// TIA Portal V15.1 export
// export: Created 2026-01-15T16:29:37.3417303Z, ExportSetting WithDefaults, WithReadOnly, DisplayName Totally Integrated Automation Portal, DisplayVersion V15.1 Update 8, DisplayName TIA Portal Openness, DisplayVersion V15.1 Update 8, DisplayName STEP 7 Professional, DisplayVersion V15.1 Update 8, DisplayName WinCC Advanced, DisplayVersion V15.1 Update 8
DATA_BLOCK "1.0 ANALOG_WAGG2"   // DB14
{ S7_Optimized_Access := 'TRUE' }
VERSION : 0.1
// stored: AutoNumber true, CodeModifiedDate 2026-01-15T16:25:52.3963656Z, CompileDate 2026-01-15T16:25:52.4020796Z, CreationDate 2026-01-15T16:22:49.8270549Z, DBAccessibleFromOPCUA true, DownloadWithoutReinit false, InstanceOfName 1.ANALOG_INPUT, InstanceOfNumber 1, InstanceOfType FB, InterfaceModifiedDate 2025-09-22T19:30:11.8403437Z, IsConsistent true, IsKnowHowProtected false, IsRetainMemResEnabled false, MemoryReserve 100, ModifiedDate 2026-01-15T16:25:52.3963656Z, ParameterModified 2025-08-30T17:31:01.4104373Z, StructureModified 2025-09-22T19:30:11.8403437Z, UDAEnableTagReadback false
"1.ANALOG_INPUT"
   // VAR_INPUT
   //    AI : Int;
   //    A_MODE : Real;
   //    ZERO : Real;
   //    SPAN : Real;
   //    BT_ZERO : Bool;
   //    BT_SPAN : Bool;
   //    B_MANUAL : Real;
   //    HMI_Manual_Trigger : Bool;
   // END_VAR
   // VAR_OUTPUT
   //    W_OUT : Real;
   //    X_OUT : Real;
   // END_VAR
   // VAR RETAIN
   //    T_AI { ExternalAccessible := 'False'; ExternalVisible := 'False'; ExternalWritable := 'False'} : Real;
   //    T_AN { ExternalAccessible := 'False'; ExternalVisible := 'False'; ExternalWritable := 'False'} : Real;
   //    T_ZERO { ExternalAccessible := 'False'; ExternalVisible := 'False'; ExternalWritable := 'False'} : Real;
   //    AN_ZERO { ExternalAccessible := 'False'; ExternalVisible := 'False'; ExternalWritable := 'False'} : Real;
   //    T_SPAN { ExternalAccessible := 'False'; ExternalVisible := 'False'; ExternalWritable := 'False'} : Real;
   //    AN_SPAN { ExternalAccessible := 'False'; ExternalVisible := 'False'; ExternalWritable := 'False'} : Real;
   // END_VAR
   // VAR
   //    B_MANUAL_SAVED : Real;
   //    B_HAS_CHANGED : Bool;
   // END_VAR
   // VAR RETAIN
   //    IS_MANUAL_MODE : Bool;
   // END_VAR
   // VAR
   //    BT_ZERO_Raising : Bool;
   //    BT_SPAN_Riasing : Bool;
   //    MANUAL_Raissing : Bool;
   //    Bit_Reset_Man_Mode : Bool;
   // END_VAR
BEGIN
END_DATA_BLOCK
